TYPE TcoIrc5_Outputs_v_1_x_x :
STRUCT
	Outputs AT %Q* : ARRAY[0..63] OF BYTE;
END_STRUCT
END_TYPE

(* stored: Version 1.1.0.1, ProductVersion 3.1.4024.12
   DUT TcoIrc5_Outputs_v_1_x_x: Id {4f05c10a-961c-0379-1a30-f2e6e821270a} *)
